PROGRAM MAIN
VAR
	pNewNode : POINTER TO Node;
	
	bCreate : BOOL := FALSE;
	bDelete: BOOL := FALSE;
END_VAR

IF bCreate AND pNewNode = 0 THEN
	pNewNode := __NEW(Node, 1);
	bCreate := FALSE;
END_IF;

IF bDelete THEN
	__DELETE(pNewNode);
	bDelete := FALSE;
END_IF

END_PROGRAM

(* stored: Version 1.1.0.1
   POU MAIN: Id {5476d895-76ae-435d-9782-f6b13de03fcd}, SpecialFunc None *)
